! Keevitus 4.5, paagi keevitus kere seest, ?lemine perimeeter, 200+480+200 mm
MoveJ [[1166.72,200.76,754.22],[0.178804,0.624372,-0.674087,0.351848],[1,-1,0,0],[1642.5,-0.000860473,-0.00206977,9E+09,9E+09,9E+09]], v600, z5, tPKI500\WObj:=w7000714;
MoveJ [[768.08,246.74,591.99],[0.154796,0.528852,-0.735934,0.393392],[1,-1,0,0],[1642.5,-10.0074,10.0282,9E+09,9E+09,9E+09]], v600, z5, tPKI500\WObj:=w7000714;
MoveJ [[714.09,147.89,358.50],[0.225232,0.837144,-0.327827,0.375489],[1,0,-1,0],[1642.5,-10.0076,10.0282,9E+09,9E+09,9E+09]], v600, z5, tPKI500\WObj:=w7000714;
ArcLStart [[728.05,133.48,311.58],[0.225215,0.837245,-0.327668,0.375413],[1,0,-1,0],[1642.5,-10.0073,10.0263,9E+09,9E+09,9E+09]], v600, seam1, m178job71, fine, tPKI500\WObj:=w7000714;
ArcL [[731.78,132.97,313.87],[0.240446,0.872935,-0.311321,0.288531],[1,0,-1,0],[1642.5,-10.0064,10.0273,9E+09,9E+09,9E+09]], v600, seam1, m178job71, z5, tPKI500\WObj:=w7000714;
ArcL [[741.60,132.83,314.58],[0.29466,0.908407,-0.270939,0.120687],[1,0,-1,0],[1642.5,-10.0074,10.0279,9E+09,9E+09,9E+09]], v600, seam1, m178job71, z5, tPKI500\WObj:=w7000714;
ArcL [[910.71,134.35,280.92],[0.294691,0.908428,-0.27085,0.120657],[0,0,-2,0],[1642.5,-10.0043,10.0255,9E+09,9E+09,9E+09]], v600, seam1, m178job71, z5, tPKI500\WObj:=w7000714;
ArcL [[922.12,135.61,281.18],[0.279875,0.895951,-0.24893,0.238699],[1,0,-1,0],[1642.5,-10.0074,10.0278,9E+09,9E+09,9E+09]], v600, seam1, m178job71, z5, tPKI500\WObj:=w7000714;
ArcLEnd [[922.62,141.92,281.42],[0.279881,0.895944,-0.248942,0.238705],[1,0,-1,0],[1642.5,-10.0074,10.0275,9E+09,9E+09,9E+09]], v600, seam1, m178job71, fine, tPKI500\WObj:=w7000714;
!
! lisatud wave
! tagant
MoveJ [[875.14,205.61,382.45],[0.279827,0.895934,-0.249016,0.238729],[1,0,-1,0],[1642.5,-10.0075,10.028,9E+09,9E+09,9E+09]], v600, z5, tPKI500\WObj:=w7000714;
! vahetada kiirust v6 v4 peale, sisemis mootori plaadi keevitus.
!Stop;
MoveJ [[865.35,316.77,434.79],[0.116074,-0.918576,0.297867,-0.232427],[1,0,-2,0],[1642.5,-10.0075,10.0279,9E+09,9E+09,9E+09]], v600, z5, tPKI500\WObj:=w7000714;
ArcLStart [[926.89,602.47,281.95],[0.171376,-0.936359,0.129511,-0.277651],[1,0,-2,0],[1642.51,-14.9733,15.0033,9E+09,9E+09,9E+09]], v600, seam1, m178job72, fine, tPKI500\WObj:=w7000714;
ArcL [[926.87,568.08,279.51],[0.00893682,-0.937691,0.124368,-0.324329],[1,0,-2,0],[1642.51,-14.9738,15.0031,9E+09,9E+09,9E+09]], v600, seam1, m178job72, z5, tPKI500\WObj:=w7000714;
ArcL [[925.93,323.18,279.50],[0.0485623,0.933539,-0.130258,0.330425],[1,0,-2,0],[1642.52,-14.972,15.0016,9E+09,9E+09,9E+09]], v600, seam1, m178job72, z5, tPKI500\WObj:=w7000714;
ArcL [[925.26,220.26,279.26],[0.0817255,0.935642,-0.127401,0.31885],[1,0,-2,0],[1642.51,-14.9732,15.0032,9E+09,9E+09,9E+09]], v600, seam1, m178job72, z5, tPKI500\WObj:=w7000714;
ArcLEnd [[923.08,136.67,281.83],[0.114078,0.93955,-0.126756,0.29693],[1,0,-2,0],[1642.51,-14.9734,15.0032,9E+09,9E+09,9E+09]], v600, seam1, m178job72, fine, tPKI500\WObj:=w7000714;
MoveJ [[835.54,241.64,426.42],[0.113929,0.939526,-0.126799,0.297043],[1,0,-2,0],[1642.51,-14.9735,15.0031,9E+09,9E+09,9E+09]], v600, z5, tPKI500\WObj:=w7000714;
!Stop;
!
!
!
!parem serv
MoveJ [[789.61,533.16,507.65],[0.224235,-0.952885,-0.0679482,-0.192649],[1,0,-2,0],[1642.51,-9.95104,-9.97571,9E+09,9E+09,9E+09]], v600, z5, tPKI500\WObj:=w7000714;
MoveJ [[647.14,569.61,433.86],[0.223791,-0.860771,-0.25761,-0.377663],[1,0,-2,0],[1642.51,-9.951,-9.97571,9E+09,9E+09,9E+09]], v600, z5, tPKI500\WObj:=w7000714;
ArcLStart [[727.96,611.07,312.95],[0.295562,-0.83914,-0.288966,-0.353535],[1,0,-2,0],[1642.51,-9.95001,-9.97452,9E+09,9E+09,9E+09]], v600, seam1, m178job71, fine, tPKI500\WObj:=w7000714;
ArcL [[732.79,610.32,317.12],[0.233775,-0.892702,-0.242611,-0.299288],[1,0,-2,0],[1642.51,-9.95127,-9.97524,9E+09,9E+09,9E+09]], v600, seam1, m178job71, z5, tPKI500\WObj:=w7000714;
ArcL [[737.79,609.46,317.60],[0.277417,-0.862841,-0.352886,-0.232418],[1,0,-2,0],[1642.51,-9.951,-9.97587,9E+09,9E+09,9E+09]], v600, seam1, m178job71, z5, tPKI500\WObj:=w7000714;
ArcL [[848.31,608.76,296.63],[0.329544,-0.875695,-0.325912,-0.135432],[1,0,-2,0],[1642.51,-9.95093,-9.97579,9E+09,9E+09,9E+09]], v600, seam1, m178job71, z5, tPKI500\WObj:=w7000714;
ArcL [[912.96,610.64,282.06],[0.338522,-0.884944,-0.249387,-0.200211],[0,0,-2,0],[1642.51,-9.95089,-9.97587,9E+09,9E+09,9E+09]], v600, seam1, m178job71, z5, tPKI500\WObj:=w7000714;
ArcLEnd [[922.77,607.32,283.12],[0.338972,-0.876763,-0.227105,-0.254579],[1,0,-2,0],[1642.51,-9.951,-9.97651,9E+09,9E+09,9E+09]], v600, seam1, m178job71, fine, tPKI500\WObj:=w7000714;
MoveJ [[629.08,382.85,564.19],[0.319673,-0.886676,-0.259097,-0.210916],[1,0,-2,0],[1642.51,-9.95097,-9.97562,9E+09,9E+09,9E+09]], v600, z5, tPKI500\WObj:=w7000714;
!Stop;
MoveJ [[687.39,482.34,438.81],[0.235271,-0.840752,-0.0361746,-0.486288],[1,0,-2,0],[1642.57,-40.0195,-20.0296,9E+09,9E+09,9E+09]], v600, z5, tPKI500\WObj:=w7000714;
MoveJ [[702.69,575.43,343.37],[0.24259,-0.815559,-0.337914,-0.40228],[1,0,-2,0],[1642.57,-40.0195,-20.0295,9E+09,9E+09,9E+09]], v600, z5, tPKI500\WObj:=w7000714;
ArcLStart [[728.60,610.74,312.98],[0.242341,-0.815698,-0.337901,-0.402159],[1,0,-2,0],[1642.57,-40.0167,-20.0299,9E+09,9E+09,9E+09]], v600, seam1, m178job71, fine, tPKI500\WObj:=w7000714;
ArcL [[720.63,611.32,299.17],[0.233436,-0.753089,-0.346163,-0.508466],[1,0,-2,0],[1642.57,-40.0193,-20.0291,9E+09,9E+09,9E+09]], v600, seam1, m178job71, z5, tPKI500\WObj:=w7000714;
ArcL [[687.24,612.19,231.30],[0.233498,-0.753121,-0.346121,-0.508418],[1,0,-2,0],[1642.57,-40.0184,-20.0296,9E+09,9E+09,9E+09]], v600, seam1, m178job71, z5, tPKI500\WObj:=w7000714;
ArcL [[665.17,611.16,193.43],[0.258577,-0.862801,-0.23332,-0.366436],[1,0,-2,0],[1642.57,-40.0177,-20.0296,9E+09,9E+09,9E+09]], v600, seam1, m178job71, z5, tPKI500\WObj:=w7000714;
ArcLEnd [[661.51,603.60,190.16],[0.237634,-0.935104,-0.126943,-0.230211],[1,1,-2,0],[1642.56,-40.0186,-20.0296,9E+09,9E+09,9E+09]], v600, seam1, m178job71, fine, tPKI500\WObj:=w7000714;
!
! lisatud wave
!paagi alumine omblus
!
MoveJ [[549.09,512.65,343.03],[0.23778,-0.935051,-0.126935,-0.230282],[1,1,-2,0],[1642.57,-40.0195,-20.0296,9E+09,9E+09,9E+09]], v600, z5, tPKI500\WObj:=w7000714;
!Stop;
MoveJ [[610.18,311.79,265.60],[0.0869508,-0.984478,-0.0404527,-0.146997],[1,1,-2,0],[1642.58,-30.2802,-29.5527,9E+09,9E+09,9E+09]], v600, z5, tPKI500\WObj:=w7000714;
ArcLStart [[661.41,139.64,189.28],[0.194623,0.960194,-0.0696521,0.18788],[1,1,-2,0],[1642.58,-30.2802,-29.5527,9E+09,9E+09,9E+09]], v600, seam1, m178job72, fine, tPKI500\WObj:=w7000714;
ArcL [[662.37,506.32,187.42],[0.0471849,0.986929,-0.072589,0.135933],[1,1,-2,0],[1642.58,-30.0157,-20.0181,9E+09,9E+09,9E+09]], v600, seam1, m178job72, z5, tPKI500\WObj:=w7000714;
ArcLEnd [[663.45,604.68,191.14],[0.105846,-0.972983,0.037102,-0.201806],[1,1,-2,0],[1642.58,-30.0163,-20.018,9E+09,9E+09,9E+09]], v600, seam1, m178job72, fine, tPKI500\WObj:=w7000714;
!
! lyhike ?mblus
MoveJ [[617.30,284.42,476.03],[0.212151,0.951515,-0.144357,0.16963],[1,1,-2,0],[1642.58,-30.0165,-20.0181,9E+09,9E+09,9E+09]], v600, z5, tPKI500\WObj:=w7000714;
!Stop;
MoveJ [[651.45,220.87,434.81],[0.264842,0.922097,-0.154916,0.235791],[1,0,-2,0],[1933.53,-34.9957,-3.2167,9E+09,9E+09,9E+09]], v600, z5, tPKI500\WObj:=w7000714;
ArcLStart [[728.67,134.77,313.36],[0.30273,0.917485,-0.0333896,0.255856],[1,0,-2,0],[1933.53,-34.9956,-3.21679,9E+09,9E+09,9E+09]], v600, seam1, m178job71, fine, tPKI500\WObj:=w7000714;
ArcL [[724.98,135.31,307.57],[0.302757,0.917479,-0.0333964,0.255845],[1,0,-2,0],[1933.53,-34.9956,-3.21658,9E+09,9E+09,9E+09]], v600, seam1, m178job71, z5, tPKI500\WObj:=w7000714;
ArcL [[671.99,137.01,206.82],[0.302795,0.91747,-0.0334103,0.255828],[1,0,-2,0],[1933.53,-34.9956,-3.21679,9E+09,9E+09,9E+09]], v600, seam1, m178job71, z5, tPKI500\WObj:=w7000714;
ArcL [[664.98,136.99,190.97],[0.302877,0.917453,-0.0334249,0.255792],[1,0,-2,0],[1933.53,-34.9956,-3.21658,9E+09,9E+09,9E+09]], v600, seam1, m178job71, z5, tPKI500\WObj:=w7000714;
ArcLEnd [[664.39,139.97,190.67],[0.302877,0.917455,-0.0334302,0.255786],[1,0,-2,0],[1933.53,-34.9957,-3.21658,9E+09,9E+09,9E+09]], v600, seam1, m178job71, fine, tPKI500\WObj:=w7000714;
MoveJ [[621.65,263.46,419.87],[0.302888,0.917449,-0.0334298,0.255793],[1,0,-2,0],[1933.53,-34.9957,-3.21658,9E+09,9E+09,9E+09]], v600, z5, tPKI500\WObj:=w7000714;

MoveJ [[1209.88,107.35,1002.71],[0.253271,0.875994,-0.262765,0.315348],[0,0,-2,0],[1642.58,-35.0333,19.9774,9E+09,9E+09,9E+09]], v600, z5, tPKI500\WObj:=w7000714;
!Stop;
! viia parandused sisse, kuumem kaar ja nurgad t?ita

! laua p??ramine -50 ja -90 kraadi
MoveJ [[463.28,65.52,1004.63],[0.457365,0.217534,-0.820402,-0.265402],[1,0,-2,0],[1642.51,-50.0165,-90.0065,9E+09,9E+09,9E+09]], v200, z5, tPKI500\WObj:=w7000714;

! Keevitus 4.6, p?hja ?mblus seest, 410+190 mm, paremalt
MoveJ [[196.38,248.72,1103.93],[0.699729,-0.625929,-0.332338,-0.0902487],[1,0,-2,0],[1642.51,-50.0165,-90.0066,9E+09,9E+09,9E+09]], v600, z5, tPKI500\WObj:=w7000714;
MoveJ [[61.15,515.96,761.72],[0.695758,-0.625539,-0.342321,-0.0862556],[1,1,-2,0],[1642.51,-50.0158,-90.0066,9E+09,9E+09,9E+09]], v600, z5, tPKI500\WObj:=w7000714;
MoveJ [[-48.26,518.22,717.52],[0.699706,-0.625962,-0.332322,-0.0902608],[1,1,-2,0],[1642.51,-50.0156,-90.0066,9E+09,9E+09,9E+09]], v600, z5, tPKI500\WObj:=w7000714;
MoveJ [[-178.59,455.25,672.83],[0.499833,-0.795207,-0.343189,0.00592692],[1,1,-2,0],[1642.51,-50.0156,-90.0066,9E+09,9E+09,9E+09]], v600, z5, tPKI500\WObj:=w7000714;
MoveJ [[-180.79,492.80,657.18],[0.521548,-0.780897,-0.342706,-0.0272303],[1,1,-2,0],[1642.51,-53.4217,-90.0073,9E+09,9E+09,9E+09]], v600, z5, tPKI500\WObj:=w7000714;
ArcLStart [[-239.25,512.85,655.67],[0.502988,-0.848154,-0.154897,0.0603867],[1,1,-3,0],[1642.51,-53.4215,-90.0079,9E+09,9E+09,9E+09]], v600, seam1, m178job73, fine, tPKI500\WObj:=w7000714;
!ArcL [[-148.87,554.55,608.87],[0.508794,-0.780118,-0.362131,0.0375068],[1,1,-2,0],[1642.51,-50.0154,-90.0066,9E+09,9E+09,9E+09]], v600, seam1, wld200v6sh14, z5, tPKI500\WObj:=w7000714;
ArcLEnd [[-35.01,617.08,549.75],[0.452558,-0.879456,-0.14001,0.0463462],[1,1,-2,0],[1642.51,-57.3737,-90.0072,9E+09,9E+09,9E+09]], v600, seam1, m178job73, fine, tPKI500\WObj:=w7000714;
MoveL [[53.79,568.86,617.64],[0.452549,-0.879461,-0.140004,0.0463546],[1,1,-2,0],[1642.51,-57.3737,-90.0073,9E+09,9E+09,9E+09]], v600, z5, tPKI500\WObj:=w7000714;
MoveJ [[35.56,572.76,595.15],[0.503916,-0.851326,-0.141306,0.0367077],[1,1,-2,0],[1642.51,-64.1768,-89.8231,9E+09,9E+09,9E+09]], v600, z5, tPKI500\WObj:=w7000714;
ArcLStart [[-26.02,618.24,544.95],[0.43508,-0.890284,-0.119141,0.0625034],[1,1,-2,0],[1642.51,-64.1769,-89.8229,9E+09,9E+09,9E+09]], v600, seam1, m178job73, fine, tPKI500\WObj:=w7000714;
ArcLEnd [[135.95,615.43,462.61],[0.421252,-0.894487,-0.14864,-0.0186384],[1,1,-2,0],[1642.51,-64.1769,-89.8228,9E+09,9E+09,9E+09]], v600, seam1, m178job73, fine, tPKI500\WObj:=w7000714;
MoveJ [[177.09,497.45,621.56],[0.421267,-0.89448,-0.148643,-0.0186307],[1,1,-2,0],[1642.51,-64.1768,-89.823,9E+09,9E+09,9E+09]], v600, z5, tPKI500\WObj:=w7000714;
!Stop;
! liiga palju t?idab, kiirust t?sta

! Keevitus 4.7, p?hja ?mblus seest, 180 mm, paremalt
MoveJ [[404.65,497.01,626.01],[0.429163,-0.845716,-0.305144,-0.0864462],[1,1,-2,0],[1950.19,-50.0155,-90.0066,9E+09,9E+09,9E+09]], v600, z5, tPKI500\WObj:=w7000714;
MoveJ [[512.35,464.70,588.20],[0.429153,-0.845719,-0.305149,-0.0864401],[1,1,-3,0],[1950.19,-50.0155,-90.0065,9E+09,9E+09,9E+09]], v600, z5, tPKI500\WObj:=w7000714;
MoveJ [[519.14,513.74,923.36],[0.398656,-0.898555,-0.0969189,-0.155823],[1,-1,0,0],[1950.19,-50.0155,-90.0065,9E+09,9E+09,9E+09]], v600, z5, tPKI500\WObj:=w7000714;
MoveJ [[461.61,590.34,346.14],[0.436335,-0.892563,-0.0806882,-0.0802135],[1,0,-1,0],[1950.19,-50.0154,-90.0063,9E+09,9E+09,9E+09]], v600, z5, tPKI500\WObj:=w7000714;
ArcLStart [[362.37,616.29,341.75],[0.405567,-0.907589,-0.0994243,-0.0437363],[1,0,-1,0],[1950.19,-50.0155,-90.0064,9E+09,9E+09,9E+09]], v600, seam1, m178job73, fine, tPKI500\WObj:=w7000714;
ArcLEnd [[521.04,611.94,261.93],[0.375808,-0.920622,-0.0997011,-0.0358339],[1,0,-1,0],[1950.19,-50.0155,-90.0071,9E+09,9E+09,9E+09]], v600, seam1, m178job73, fine, tPKI500\WObj:=w7000714;
MoveJ [[520.88,573.24,288.35],[0.346336,-0.937403,-0.0309934,-0.0191679],[1,0,-1,0],[1912.44,-50.0155,-90.0084,9E+09,9E+09,9E+09]], v600, z5, tPKI500\WObj:=w7000714;
ArcLStart [[531.51,613.38,255.56],[0.346292,-0.937416,-0.0310979,-0.0191738],[1,0,-1,0],[1912.44,-50.0155,-90.0083,9E+09,9E+09,9E+09]], v600, seam1, m178job73, fine, tPKI500\WObj:=w7000714;
ArcLEnd [[653.72,608.94,194.33],[0.390845,-0.857992,-0.281743,-0.178077],[1,0,0,0],[1959.61,-55.9377,-89.965,9E+09,9E+09,9E+09]], v600, seam1, m178job73, fine, tPKI500\WObj:=w7000714;
MoveL [[657.28,415.67,487.92],[0.390843,-0.857996,-0.281742,-0.178065],[1,-1,0,0],[1959.61,-55.9377,-89.9649,9E+09,9E+09,9E+09]], v600, z5, tPKI500\WObj:=w7000714;

GOTO paagiall;

! Keevitus 4.8, paagi ?mblus seest, ?lalt-alla, 150 mm, paremalt
MoveJ [[708.82,589.48,349.92],[0.26351,-0.882482,-0.294377,-0.25521],[1,1,-2,0],[1950.19,-50.0147,-90.0062,9E+09,9E+09,9E+09]], v600, z5, tPKI500\WObj:=w7000714;
ArcLStart [[732.29,612.15,312.42],[0.263422,-0.882509,-0.294419,-0.255159],[1,1,-2,0],[1950.19,-50.0147,-90.0062,9E+09,9E+09,9E+09]], v600, seam1, wld100v4sh16, fine, tPKI500\WObj:=w7000714;
ArcL [[721.14,612.59,306.41],[0.263365,-0.882522,-0.294466,-0.255117],[1,1,-2,0],[1950.19,-50.0148,-90.0059,9E+09,9E+09,9E+09]], v600, seam1, wld100v4sh16, z5, tPKI500\WObj:=w7000714;
ArcLEnd [[660.86,607.69,192.53],[0.282267,-0.873646,-0.270174,-0.289957],[1,1,-2,0],[1950.19,-50.0148,-90.0062,9E+09,9E+09,9E+09]], v600, seam1, wld100v4sh16, fine, tPKI500\WObj:=w7000714;
MoveJ [[659.87,534.23,289.89],[0.282313,-0.873638,-0.270157,-0.289951],[1,1,-2,0],[1950.19,-50.0147,-90.0062,9E+09,9E+09,9E+09]], v600, z5, tPKI500\WObj:=w7000714;
MoveJ [[656.91,166.38,784.04],[0.282307,-0.87364,-0.27016,-0.289949],[1,0,-1,0],[1950.19,-50.0147,-90.0062,9E+09,9E+09,9E+09]], v600, z5, tPKI500\WObj:=w7000714;
MoveJ [[655.16,-102.11,1008.14],[0.282304,-0.87364,-0.27016,-0.289954],[1,0,-1,0],[1950.19,-50.0147,-90.0061,9E+09,9E+09,9E+09]], v600, z5, tPKI500\WObj:=w7000714;
! liiga palju t?idab, kiirust t?sta

paagiall:

! laua p??ramine 50 ja -90 kraadi
MoveJ [[629.05,106.87,1333.63],[0.742615,-0.0488617,-0.662818,0.0825176],[1,0,-2,0],[1950.19,-50.0144,-90.0065,9E+09,9E+09,9E+09]], v600, z5, tPKI500\WObj:=w7000714;
MoveJ [[666.24,1407.62,346.58],[0.485843,0.779341,0.394853,-0.0260103],[1,0,-1,0],[1950.2,49.9779,-90.0059,9E+09,9E+09,9E+09]], v200, z5, tPKI500\WObj:=w7000714;

! Keevitus 4.9, p?hja ?mblus seest, 410+190 mm, vasakult
MoveJ [[388.60,678.79,1213.60],[0.557133,0.824872,0.0604223,0.0744247],[0,0,-1,0],[12.7994,49.9779,-90.0058,9E+09,9E+09,9E+09]], v600, z5, tPKI500\WObj:=w7000714;
MoveJ [[384.49,294.23,786.50],[0.557145,0.824863,0.0604211,0.074436],[0,0,-1,0],[12.7984,49.978,-90.0056,9E+09,9E+09,9E+09]], v600, z5, tPKI500\WObj:=w7000714;
MoveJ [[65.60,161.93,784.24],[0.484927,0.853835,-0.0416443,-0.184603],[0,1,-2,0],[12.7988,49.978,-90.0056,9E+09,9E+09,9E+09]], v600, z5, tPKI500\WObj:=w7000714;
MoveJ [[-229.88,281.25,701.83],[0.48494,0.85383,-0.0416313,-0.184598],[0,1,-2,0],[12.7988,49.978,-90.0056,9E+09,9E+09,9E+09]], v600, z5, tPKI500\WObj:=w7000714;
ArcLStart [[-229.82,242.03,655.30],[0.485298,0.853687,-0.0412593,-0.184401],[0,1,-2,0],[12.7994,49.9782,-90.0049,9E+09,9E+09,9E+09]], v600, seam1, m178job75, fine, tPKI500\WObj:=w7000714;
ArcL [[-84.08,165.89,578.50],[0.498551,0.849644,-0.0346232,-0.16839],[0,1,-2,0],[12.7972,49.9796,-90.004,9E+09,9E+09,9E+09]], v600, seam1, m178job75, z5, tPKI500\WObj:=w7000714;
ArcL [[-27.66,140.23,549.05],[0.527487,0.84556,-0.00876734,-0.0819137],[0,1,-2,0],[12.7972,49.9795,-90.0041,9E+09,9E+09,9E+09]], v600, seam1, m178job75, z5, tPKI500\WObj:=w7000714;
ArcL [[16.72,138.82,525.36],[0.481758,0.871608,-0.0848704,-0.0317208],[0,1,-2,0],[12.7933,49.9797,-90.0036,9E+09,9E+09,9E+09]], v600, seam1, m178job75, z5, tPKI500\WObj:=w7000714;
ArcLEnd [[133.70,138.04,464.64],[0.451188,0.883091,-0.127052,0.0209757],[0,2,-2,0],[12.7949,49.9799,-90.0038,9E+09,9E+09,9E+09]], v600, seam1, m178job73, fine, tPKI500\WObj:=w7000714;
MoveJ [[136.36,209.25,580.64],[0.468487,0.870946,-0.136243,-0.0584185],[0,1,-2,0],[12.7984,49.978,-90.0055,9E+09,9E+09,9E+09]], v600, z5, tPKI500\WObj:=w7000714;
! liiga palju t?idab, kiirust t?sta

! Keevitus 4.10, sarniiri k?rv pealt, 100+50, vasakult
MoveJ [[-36.62,215.87,637.30],[0.532452,0.822587,-0.164204,-0.113512],[0,1,-2,0],[12.8001,49.9781,-90.0053,9E+09,9E+09,9E+09]], v600, z5, tPKI500\WObj:=w7000714;
ArcLStart [[-77.82,169.87,614.91],[0.492202,0.845085,-0.126744,-0.165852],[0,1,-2,0],[12.8004,49.9783,-90.0044,9E+09,9E+09,9E+09]], v600, seam1, m178job75, fine, tPKI500\WObj:=w7000714;
ArcL [[-14.48,137.24,582.80],[0.468789,0.86953,-0.05854,-0.143978],[0,1,-2,0],[12.8017,49.9785,-90.005,9E+09,9E+09,9E+09]], v600, seam1, m178job75, z5, tPKI500\WObj:=w7000714;
ArcLEnd [[24.32,136.30,561.78],[0.4688,0.869526,-0.0585137,-0.143972],[0,1,-2,0],[12.8017,49.9783,-90.0048,9E+09,9E+09,9E+09]], v600, seam1, m178job75, fine, tPKI500\WObj:=w7000714;
MoveJ [[26.28,211.80,629.17],[0.53258,0.822524,-0.164103,-0.11351],[0,1,-2,0],[12.8001,49.9781,-90.0056,9E+09,9E+09,9E+09]], v600, z5, tPKI500\WObj:=w7000714;
MoveJ [[454.07,297.49,698.34],[0.532584,0.822521,-0.164102,-0.113513],[0,1,-2,0],[12.8001,49.978,-90.0054,9E+09,9E+09,9E+09]], v600, z5, tPKI500\WObj:=w7000714;
! liiga kuum

! Keevitus 4.11, p?hja ?mblus seest, 180 mm, vasakult
MoveJ [[462.46,181.06,454.07],[0.532569,0.822509,-0.164117,-0.113651],[0,1,-2,0],[12.7994,49.9781,-90.0054,9E+09,9E+09,9E+09]], v600, z5, tPKI500\WObj:=w7000714;
MoveJ [[373.51,148.16,352.75],[0.532701,0.836564,-0.127494,0.0116893],[0,1,-2,0],[12.8004,49.9782,-90.0053,9E+09,9E+09,9E+09]], v600, z5, tPKI500\WObj:=w7000714;
ArcLStart [[363.62,133.40,339.74],[0.385285,0.913722,-0.128687,-0.0104206],[0,1,-3,0],[12.8033,49.9784,-90.0053,9E+09,9E+09,9E+09]], v600, seam1, m178job73, fine, tPKI500\WObj:=w7000714;
ArcLEnd [[521.63,134.33,258.78],[0.384893,0.913779,-0.129338,-0.0118155],[0,1,-2,0],[12.804,49.978,-90.0048,9E+09,9E+09,9E+09]], v600, seam1, m178job73, fine, tPKI500\WObj:=w7000714;
MoveJ [[529.89,336.50,401.69],[0.385019,0.91381,-0.12889,-0.00995835],[0,1,-2,0],[12.8004,49.9781,-90.0051,9E+09,9E+09,9E+09]], v600, z5, tPKI500\WObj:=w7000714;
MoveJ [[533.43,251.88,352.38],[0.378148,0.919534,-0.10133,0.0345688],[0,1,-2,0],[12.8017,49.9784,-90.005,9E+09,9E+09,9E+09]], v600, z5, tPKI500\WObj:=w7000714;
ArcLStart [[531.13,134.57,252.75],[0.378146,0.919534,-0.101345,0.0345315],[0,1,-2,0],[12.8017,49.9784,-90.005,9E+09,9E+09,9E+09]], v600, seam1, m178job73, fine, tPKI500\WObj:=w7000714;
ArcLEnd [[657.61,136.14,189.32],[0.303811,0.940087,-0.0293689,0.151901],[0,1,-3,0],[12.7988,49.9785,-90.0046,9E+09,9E+09,9E+09]], v600, seam1, m178job73, fine, tPKI500\WObj:=w7000714;
MoveL [[549.64,239.77,442.99],[0.323521,0.93805,-0.0571311,0.110153],[0,1,-3,0],[12.7994,49.9786,-90.005,9E+09,9E+09,9E+09]], v600, z5, tPKI500\WObj:=w7000714;

MoveJ [[730.99,435.16,896.64],[0.414132,0.875986,-0.0952889,0.228177],[0,-1,0,0],[12.8004,49.9782,-90.0052,9E+09,9E+09,9E+09]], v600, z5, tPKI500\WObj:=w7000714;
MoveJ [[630.56,205.75,1267.74],[0.0352222,0.637589,0.698102,-0.323875],[1,0,-2,0],[63.5912,90.0341,-90.0151,9E+09,9E+09,9E+09]], v600, z5, tPKI500\WObj:=w7000714;

! laua p??ramine 90 ja -90 kraadi
MoveJ [[628.71,206.23,996.67],[0.0352126,0.637586,0.698102,-0.32388],[1,0,-2,0],[334.665,90.0341,-90.0152,9E+09,9E+09,9E+09]], v200, z5, tPKI500\WObj:=w7000714;
MoveJ [[897.19,986.56,937.18],[0.846952,0.13011,-0.222738,0.464901],[1,-1,1,0],[1328.03,90.034,-90.0145,9E+09,9E+09,9E+09]], v200, z5, tPKI500\WObj:=w7000714;
MoveJ [[1264.54,861.62,340.94],[0.846954,0.130102,-0.222719,0.464908],[1,-1,2,0],[1328.03,90.0341,-90.0147,9E+09,9E+09,9E+09]], v200, z5, tPKI500\WObj:=w7000714;

! Keevitus 4.19, tagumine kereplaat, l?hike ?mblus, 30 mm, paremalt, OK
MoveJ [[1033.09,580.58,354.82],[0.686293,0.0368718,-0.42949,-0.585817],[1,-1,-1,0],[2188.28,-90.0189,-90.0141,9E+09,9E+09,9E+09]], v600, z5, tPKI500\WObj:=w7000714;
MoveJ [[979.14,569.48,388.43],[0.806601,-0.0278027,-0.197946,-0.556273],[1,-1,0,0],[2188.28,-90.0189,-90.0141,9E+09,9E+09,9E+09]], v600, z5, tPKI500\WObj:=w7000714;
ArcLStart [[978.92,568.70,409.45],[0.806531,-0.0276883,-0.198257,-0.55627],[1,-1,0,0],[2188.28,-90.0187,-90.0134,9E+09,9E+09,9E+09]], v600, seam1, m178job74, fine, tPKI500\WObj:=w7000714;
ArcLEnd [[979.79,595.48,407.03],[0.806541,-0.0276795,-0.198221,-0.556269],[1,-1,0,0],[2188.28,-90.0191,-90.0136,9E+09,9E+09,9E+09]], v600, seam1, m178job74, fine, tPKI500\WObj:=w7000714;
MoveL [[991.84,562.72,392.18],[0.806551,-0.0277066,-0.198182,-0.556268],[1,-1,0,0],[2188.28,-90.0181,-90.0139,9E+09,9E+09,9E+09]], v600, z5, tPKI500\WObj:=w7000714;
MoveJ [[984.53,239.20,388.90],[0.844678,0.202999,-0.0676416,-0.49065],[1,-1,-1,0],[2188.28,-90.0188,-90.0142,9E+09,9E+09,9E+09]], v600, z5, tPKI500\WObj:=w7000714;
ArcLStart [[975.41,149.41,410.22],[0.844693,0.203001,-0.0678212,-0.490598],[1,-1,-1,0],[2188.28,-90.018,-90.0166,9E+09,9E+09,9E+09]], v600, seam1, m178job74, fine, tPKI500\WObj:=w7000714;
ArcLEnd [[974.88,173.69,411.07],[0.844673,0.203034,-0.0678784,-0.49061],[1,-1,-1,0],[2188.28,-90.0188,-90.0144,9E+09,9E+09,9E+09]], v600, seam1, m178job74, fine, tPKI500\WObj:=w7000714;
MoveJ [[1127.32,173.99,318.93],[0.844677,0.203007,-0.0677125,-0.490637],[1,-1,-1,0],[2188.28,-90.0188,-90.0143,9E+09,9E+09,9E+09]], v600, z5, tPKI500\WObj:=w7000714;
MoveJ [[1123.72,259.36,389.60],[0.806585,-0.0277724,-0.198013,-0.556274],[1,-1,-1,0],[2188.28,-90.0189,-90.014,9E+09,9E+09,9E+09]], v600, z5, tPKI500\WObj:=w7000714;
MoveJ [[1120.90,-120.19,388.59],[0.806586,-0.0277689,-0.198012,-0.556274],[1,-1,-1,0],[2188.28,-90.019,-90.014,9E+09,9E+09,9E+09]], v600, z5, tPKI500\WObj:=w7000714;
MoveJ [[1027.41,-315.13,387.66],[0.806588,-0.0277633,-0.198009,-0.556273],[1,-1,-1,0],[2188.28,-90.019,-90.0141,9E+09,9E+09,9E+09]], v600, z5, tPKI500\WObj:=w7000714;
MoveJ [[1587.39,-314.57,2238.78],[0.395106,-0.543248,0.72299,-0.16143],[0,-1,-1,0],[2188.28,-90.0189,-90.0141,9E+09,9E+09,9E+09]], v600, z5, tPKI500\WObj:=w7000714;

! laua p??ramine 0 ja 0 kraadi
MoveJ [[2571.99,-849.77,725.34],[0.516673,0.188187,-0.752202,0.36308],[0,-1,-1,0],[2188.28,-0.0178089,-0.0101717,9E+09,9E+09,9E+09]], v200, z5, tPKI500\WObj:=w7000714;
MoveJ [[1078.51,394.47,809.90],[0.143804,-0.871177,0.456961,-0.107516],[1,-1,0,0],[2188.28,-0.0178089,-0.0101295,9E+09,9E+09,9E+09]], v600, z5, tPKI500\WObj:=w7000714;
MoveL [[784.81,404.00,996.38],[0.219819,-0.844688,0.418448,-0.251165],[1,-1,0,0],[2188.28,-19.3919,-1.07477,9E+09,9E+09,9E+09]], v600, z5, tPKI500\WObj:=w7000714;
MoveL [[830.09,498.09,533.40],[0.157013,-0.745399,0.376549,-0.5272],[1,-1,0,0],[2188.28,-33.0668,-1.07519,9E+09,9E+09,9E+09]], v600, z5, tPKI500\WObj:=w7000714;
ArcLStart [[968.89,134.51,399.97],[0.229202,0.70512,-0.224113,0.632493],[1,0,-1,0],[2188.27,-33.0655,-1.07654,9E+09,9E+09,9E+09]], v200, seam1, m178job77, fine, tPKI500\WObj:=w7000714;
ArcL [[932.09,135.02,326.61],[0.229208,0.705135,-0.224106,0.632476],[1,0,-1,0],[2188.27,-33.0655,-1.07633,9E+09,9E+09,9E+09]], v200, seam1, m178job77, fine, tPKI500\WObj:=w7000714;
ArcL [[924.27,137.56,288.65],[0.285048,0.869977,-0.140228,0.377128],[1,0,-2,0],[2188.27,-33.0647,-1.07713,9E+09,9E+09,9E+09]], v200, seam1, m178job77, fine, tPKI500\WObj:=w7000714;
ArcLEnd [[916.79,146.87,290.75],[0.225012,0.93026,-0.175906,0.230313],[1,1,-2,0],[2188.27,-33.0647,-1.07692,9E+09,9E+09,9E+09]], v200, seam1, m178job77, fine, tPKI500\WObj:=w7000714;
MoveL [[860.28,390.12,368.97],[0.0097858,0.933264,-0.105499,0.343212],[1,0,-2,0],[2188.27,-33.0647,-1.07705,9E+09,9E+09,9E+09]], v200, fine, tPKI500\WObj:=w7000714;
ArcLStart [[966.40,607.71,401.95],[0.309024,-0.838606,-0.190201,-0.406287],[1,0,-2,0],[2188.27,-33.0639,-1.07755,9E+09,9E+09,9E+09]], v200, seam1, m178job77, fine, tPKI500\WObj:=w7000714;
ArcL [[930.19,608.39,328.98],[0.308956,-0.838652,-0.190164,-0.406262],[1,0,-2,0],[2188.27,-33.0639,-1.07776,9E+09,9E+09,9E+09]], v200, seam1, m178job77, fine, tPKI500\WObj:=w7000714;
ArcL [[923.99,606.70,286.47],[0.284962,-0.883566,-0.155473,-0.337548],[1,1,-2,0],[2188.27,-33.0634,-1.07882,9E+09,9E+09,9E+09]], v200, seam1, m178job77, fine, tPKI500\WObj:=w7000714;
ArcLEnd [[922.74,604.55,283.86],[0.225597,-0.927343,-0.17685,-0.240556],[1,1,-2,0],[2188.27,-33.0634,-1.07882,9E+09,9E+09,9E+09]], v200, seam1, m178job77, fine, tPKI500\WObj:=w7000714;
MoveL [[766.07,413.97,534.40],[0.285128,-0.883476,-0.155522,-0.337618],[1,0,-2,0],[2188.27,-33.0637,-1.07827,9E+09,9E+09,9E+09]], v600, fine, tPKI500\WObj:=w7000714;
MoveL [[1931.24,112.08,1797.85],[0.481099,-0.603835,0.414467,-0.481815],[0,0,-2,0],[2188.27,-33.0635,-1.07827,9E+09,9E+09,9E+09]], v600, fine, tPKI500\WObj:=w7000714;
! laua p??ramine 0 ja 180 kraadi
!MoveJ [[-1805.19,1600.36,726.17],[0.363056,-0.752319,-0.188029,-0.516579],[0,-1,-1,0],[2188.34,-0.0394387,180.004,9E+09,9E+09,9E+09]], v500, z5, tPKI500\WObj:=w7000714;
! laua p??ramine -40 ja 180 kraadi
!MoveJ [[-842.65,1593.50,1984.19],[0.407518,-0.88328,-0.0499407,-0.226392],[0,-1,-1,0],[2188.34,-40.3394,179.976,9E+09,9E+09,9E+09]], v200, z5, tPKI500\WObj:=w7000714;
!MoveJ [[-361.88,238.65,1366.99],[0.233905,-0.220588,-0.921934,0.216031],[0,0,-2,0],[2188.34,-34.9738,179.976,9E+09,9E+09,9E+09]], v600, z5, tPKI500\WObj:=w7000714;
!MoveJ [[-329.76,347.68,853.85],[0.171568,-0.037775,-0.971091,0.161622],[0,1,-2,0],[2188.34,-33.8713,179.976,9E+09,9E+09,9E+09]], v600, z5, tPKI500\WObj:=w7000714;
!ArcLStart [[-267.00,283.63,772.23],[0.159657,0.0398007,-0.944889,0.283041],[1,1,-2,0],[2188.34,-33.8711,179.976,9E+09,9E+09,9E+09]], v600, seam1, wld100v4sh16, fine, tPKI500\WObj:=w7000714;
!ArcLEnd [[-319.65,311.33,800.44],[0.159636,0.0398197,-0.944893,0.283035],[1,1,-2,0],[2188.34,-33.8713,179.976,9E+09,9E+09,9E+09]], v600, seam1, wld100v4sh16, fine, tPKI500\WObj:=w7000714;
!ArcLStart [[-267.16,284.07,771.57],[0.159658,0.0398083,-0.944881,0.283064],[1,1,-2,0],[2188.34,-33.871,179.976,9E+09,9E+09,9E+09]], v600, seam1, wld100v4sh16\Weave:=weave4, fine, tPKI500\WObj:=w7000714;
!ArcLEnd [[-321.12,312.86,800.70],[0.159639,0.0398143,-0.944893,0.283037],[1,1,-2,0],[2188.34,-33.8713,179.976,9E+09,9E+09,9E+09]], v600, seam1, wld100v4sh16\Weave:=weave4, fine, tPKI500\WObj:=w7000714;
!MoveL [[-422.53,369.77,925.81],[0.146248,0.0635872,-0.986461,-0.0382709],[0,0,-2,0],[2188.34,-33.8712,179.976,9E+09,9E+09,9E+09]], v600, fine, tPKI500\WObj:=w7000714;
!MoveL [[-371.17,402.53,866.35],[0.159991,-0.0776618,-0.933329,-0.311882],[0,0,-2,0],[2188.34,-33.8712,179.976,9E+09,9E+09,9E+09]], v600, fine, tPKI500\WObj:=w7000714;
!ArcLStart [[-264.44,468.19,771.49],[0.202364,-0.212347,-0.926323,-0.236398],[1,0,-2,0],[2188.34,-33.8711,179.976,9E+09,9E+09,9E+09]], v600, seam1, wld100v4sh16, fine, tPKI500\WObj:=w7000714;
!ArcLEnd [[-317.75,442.56,798.65],[0.20235,-0.212334,-0.926323,-0.236423],[1,0,-2,0],[2188.34,-33.8711,179.976,9E+09,9E+09,9E+09]], v600, seam1, wld100v4sh16, fine, tPKI500\WObj:=w7000714;
!ArcLStart [[-265.35,467.62,772.88],[0.20236,-0.212345,-0.926325,-0.236395],[1,0,-2,0],[2188.34,-33.8711,179.976,9E+09,9E+09,9E+09]], v600, seam1, wld100v4sh16\Weave:=weave4, fine, tPKI500\WObj:=w7000714;
!ArcLEnd [[-318.74,440.66,800.16],[0.202349,-0.212327,-0.926327,-0.236414],[1,0,-2,0],[2188.34,-33.871,179.976,9E+09,9E+09,9E+09]], v600, seam1, wld100v4sh16\Weave:=weave4, fine, tPKI500\WObj:=w7000714;
!MoveL [[-386.39,410.04,858.22],[0.20235,-0.21233,-0.926323,-0.236427],[0,0,-2,0],[2188.34,-33.8711,179.976,9E+09,9E+09,9E+09]], v600, fine, tPKI500\WObj:=w7000714;
!MoveJ [[-350.68,416.29,1470.07],[0.202358,-0.212326,-0.92632,-0.236433],[0,0,-1,0],[2188.34,-33.8711,179.976,9E+09,9E+09,9E+09]], v600, fine, tPKI500\WObj:=w7000714;
MoveJ [[2571.99,-849.77,725.34],[0.516675,0.188183,-0.752204,0.363076],[0,-1,-1,0],[2188.28,-0.0178089,-0.0101717,9E+09,9E+09,9E+09]], v400, fine, tPKI500\WObj:=w7000714;



! aeg manualis 15:30, 100 % juures


MoveJ mooduli_vahetus, v600, z50, tPKI500\WObj:=w7000714;

ENDPROC


! V?ljast kinnitused ja alt puksid
PROC Seest_alt()

MoveJ mooduli_vahetus, v600, z50, tPKI500\WObj:=w7000714;

!laua liikumine
!Stop;
! Keevitus 5.1, esimene vasak klots ulevalt ja korvalt.
MoveJ [[-290.14,770.26,1028.88],[0.179367,-0.475167,0.667996,-0.5439],[0,0,-1,0],[1372.29,-65.3529,37.4059,9E+09,9E+09,9E+09]], v200, z50, tPKI500\WObj:=w7000714;
MoveJ [[-43.63,789.96,1015.82],[0.0154596,0.0805408,0.981036,-0.175623],[0,-1,0,0],[1372.29,-65.3519,37.4059,9E+09,9E+09,9E+09]], v600, z50, tPKI500\WObj:=w7000714;
ArcLStart [[-30.35,722.48,992.87],[0.0308617,0.0919503,-0.954938,0.280513],[0,0,0,0],[1372.28,-65.3461,37.4041,9E+09,9E+09,9E+09]], v600, seam1, m178job76, fine, tPKI500\WObj:=w7000714;
ArcL [[4.24,779.21,976.32],[0.031198,0.0916798,-0.954822,0.280957],[0,0,0,0],[1372.3,-65.3486,37.4052,9E+09,9E+09,9E+09]], v600, seam1, m178job76, z50, tPKI500\WObj:=w7000714;
ArcL [[4.75,783.75,972.21],[0.163165,0.328816,-0.70964,0.60139],[0,0,-1,0],[1372.29,-65.3489,37.4059,9E+09,9E+09,9E+09]], v600, seam1, m178job76, z50, tPKI500\WObj:=w7000714;
ArcL [[-106.57,785.87,753.86],[0.206514,0.412137,-0.564809,0.684461],[1,0,-1,0],[1372.28,-65.3395,37.4003,9E+09,9E+09,9E+09]], v600, seam1, m178job76, z50, tPKI500\WObj:=w7000714;
ArcL [[-111.66,783.39,751.13],[0.0614244,0.527208,-0.229631,0.815812],[1,0,-1,0],[1372.28,-65.3501,37.4051,9E+09,9E+09,9E+09]], v600, seam1, m178job76, z50, tPKI500\WObj:=w7000714;
ArcLEnd [[-145.83,729.02,766.75],[0.118602,0.614006,-0.031797,0.779692],[1,0,-2,0],[1372.29,-65.3478,37.4021,9E+09,9E+09,9E+09]], v600, seam1, m178job76, fine, tPKI500\WObj:=w7000714;
MoveJ [[-215.14,772.76,801.30],[0.102061,0.714158,0.0425608,0.691196],[1,0,-2,0],[1372.29,-65.3521,37.4058,9E+09,9E+09,9E+09]], v600, z50, tPKI500\WObj:=w7000714;
MoveJ [[-208.50,762.42,1040.05],[0.137789,-0.773479,0.148928,-0.600471],[0,0,-2,0],[1372.29,-65.3521,37.4056,9E+09,9E+09,9E+09]], v600, z50, tPKI500\WObj:=w7000714;
ArcLStart [[-30.79,723.95,992.18],[0.136855,-0.804117,0.0864458,-0.57201],[0,0,-2,0],[1372.29,-65.3435,37.4035,9E+09,9E+09,9E+09]], v600, seam1, m178job76, fine, tPKI500\WObj:=w7000714;
ArcLEnd [[-145.93,726.55,773.14],[0.136768,-0.804096,0.0862477,-0.57209],[0,0,-2,0],[1372.29,-65.3446,37.4062,9E+09,9E+09,9E+09]], v600, seam1, m178job76, fine, tPKI500\WObj:=w7000714;
MoveJ [[-373.93,893.47,896.85],[0.138032,-0.80362,0.0855156,-0.572565],[0,0,-2,0],[1372.29,-65.3521,37.4057,9E+09,9E+09,9E+09]], v600, z50, tPKI500\WObj:=w7000714;




! Keevitus 5.3, p?rkeraua klots parem, esimene ?mblus, pealt ja kuljelt
MoveJ [[-174.00,-345.05,357.08],[0.250849,-0.133618,-0.812081,-0.509653],[1,0,-2,0],[1372.29,-65.4717,-36.1497,9E+09,9E+09,9E+09]], v200, z50, tPKI500\WObj:=w7000714;
MoveJ [[-10.19,-84.76,986.05],[0.275118,-0.267366,-0.642243,-0.66359],[0,0,-2,0],[1372.29,-65.4717,-36.1497,9E+09,9E+09,9E+09]], v600, z50, tPKI500\WObj:=w7000714;
ArcLStart [[-5.29,-25.23,972.07],[0.269578,-0.358495,-0.567203,-0.690718],[0,0,-2,0],[1372.33,-65.4684,-36.1495,9E+09,9E+09,9E+09]], v600, seam1, m178job76, fine, tPKI500\WObj:=w7000714;
ArcL [[-118.04,-25.80,755.94],[0.253515,-0.440375,-0.485319,-0.711524],[1,0,-2,0],[1372.28,-65.4664,-36.1515,9E+09,9E+09,9E+09]], v600, seam1, m178job76, z50, tPKI500\WObj:=w7000714;
ArcL [[-122.46,-23.08,751.12],[0.364637,-0.582226,0.0124595,-0.726566],[1,0,-1,0],[1372.3,-65.4709,-36.1507,9E+09,9E+09,9E+09]], v600, seam1, m178job76, z50, tPKI500\WObj:=w7000714;
ArcL [[-153.48,32.59,768.13],[0.37674,-0.591162,0.132537,-0.700736],[1,0,-1,0],[1372.29,-65.4696,-36.1466,9E+09,9E+09,9E+09]], v600, seam1, m178job76, z50, tPKI500\WObj:=w7000714;
ArcL [[-152.80,36.92,774.93],[0.372014,-0.520105,0.662343,-0.390384],[1,-1,0,0],[1372.29,-65.4622,-36.1483,9E+09,9E+09,9E+09]], v600, seam1, m178job76, z50, tPKI500\WObj:=w7000714;
ArcL [[-39.28,36.72,991.14],[0.345262,-0.453792,0.773924,-0.275519],[1,-1,0,0],[1372.3,-65.4589,-36.1523,9E+09,9E+09,9E+09]], v600, seam1, m178job76, z50, tPKI500\WObj:=w7000714;
ArcL [[-35.16,32.79,991.93],[0.248259,-0.27299,0.925404,0.0864419],[1,-1,0,0],[1372.28,-65.4618,-36.1461,9E+09,9E+09,9E+09]], v600, seam1, m178job76, z50, tPKI500\WObj:=w7000714;
ArcLEnd [[-4.28,-21.64,975.36],[0.137343,-0.249955,0.927968,0.239868],[1,-1,1,0],[1372.29,-65.4709,-36.1483,9E+09,9E+09,9E+09]], v600, seam1, m178job76, fine, tPKI500\WObj:=w7000714;
MoveJ [[-61.03,-65.95,1001.68],[0.133904,-0.241825,0.927325,0.252308],[1,-1,1,0],[1372.29,-65.4722,-36.1495,9E+09,9E+09,9E+09]], v600, z50, tPKI500\WObj:=w7000714;


! Keevitus 5.4, p?rkeraua klots paremalt, teine ?mblus, kuljelt.


! Keevitus 5.5, p?rkeraua klots tagant1, O ?mblus, vasakult
MoveJ [[1208.50,-67.48,645.00],[0.55081,-0.741965,0.19537,0.328526],[0,-1,0,0],[1289.08,-105.992,-131.558,9E+09,9E+09,9E+09]], v200, z50, tPKI500\WObj:=w7000714;
MoveJ [[878.05,-71.80,532.67],[0.377928,-0.771852,0.343338,0.378859],[0,-1,0,0],[1289.08,-105.992,-131.558,9E+09,9E+09,9E+09]], v600, z50, tPKI500\WObj:=w7000714;
ArcLStart [[911.48,1.66,499.56],[0.180122,-0.806357,0.321968,0.462258],[0,-1,1,0],[1289.09,-105.99,-131.558,9E+09,9E+09,9E+09]], v600, seam1, m178job76, fine, tPKI500\WObj:=w7000714;
ArcL [[866.81,-37.76,522.04],[0.241931,-0.80225,0.32882,0.435596],[0,-1,0,0],[1289.08,-105.992,-131.558,9E+09,9E+09,9E+09]], v600, seam1, m178job76, z50, tPKI500\WObj:=w7000714;
ArcL [[859.31,-43.24,520.79],[0.656383,-0.696913,0.229608,0.175374],[0,-1,0,0],[1289.08,-105.991,-131.558,9E+09,9E+09,9E+09]], v600, seam1, m178job76, z50, tPKI500\WObj:=w7000714;
ArcL [[749.03,-43.15,305.63],[0.666588,-0.691289,0.223493,0.16683],[1,-1,0,0],[1289.08,-105.991,-131.558,9E+09,9E+09,9E+09]], v600, seam1, m178job76, z50, tPKI500\WObj:=w7000714;
ArcL [[748.23,-38.21,296.26],[0.881837,-0.46223,0.0260185,-0.0896109],[1,0,-1,0],[1289.08,-105.992,-131.558,9E+09,9E+09,9E+09]], v600, seam1, m178job76, z50, tPKI500\WObj:=w7000714;
ArcLEnd [[795.12,2.54,270.09],[0.92494,-0.290166,-0.143809,-0.199024],[1,0,-1,0],[1289.08,-105.991,-131.558,9E+09,9E+09,9E+09]], v600, seam1, m178job76, fine, tPKI500\WObj:=w7000714;
MoveL [[821.17,-27.30,258.63],[0.924935,-0.290173,-0.143812,-0.199036],[1,0,-1,0],[1289.08,-105.991,-131.558,9E+09,9E+09,9E+09]], v400, z50, tPKI500\WObj:=w7000714;
MoveL [[823.25,-19.25,258.87],[0.774205,0.152692,-0.382226,-0.480829],[1,0,-2,0],[1289.08,-105.991,-131.56,9E+09,9E+09,9E+09]], v400, z50, tPKI500\WObj:=w7000714;
ArcLStart [[801.74,5.40,268.33],[0.774207,0.152706,-0.382226,-0.480821],[1,0,-2,0],[1289.08,-105.991,-131.56,9E+09,9E+09,9E+09]], v600, seam1, m178job76, fine, tPKI500\WObj:=w7000714;
ArcL [[805.46,3.98,276.41],[0.77421,0.152731,-0.382224,-0.480811],[1,0,-2,0],[1289.08,-105.992,-131.559,9E+09,9E+09,9E+09]], v600, seam1, m178job76, z50, tPKI500\WObj:=w7000714;
ArcLEnd [[913.95,3.05,493.11],[0.74603,0.191483,-0.397811,-0.498518],[0,0,-2,0],[1289.08,-105.991,-131.558,9E+09,9E+09,9E+09]], v600, seam1, m178job76, fine, tPKI500\WObj:=w7000714;
MoveJ [[1036.00,-137.14,436.44],[0.829926,0.0635067,-0.342982,-0.435379],[0,0,-2,0],[1289.08,-105.992,-131.558,9E+09,9E+09,9E+09]], v600, z50, tPKI500\WObj:=w7000714;
MoveJ [[771.13,-196.57,635.64],[0.451534,0.540448,-0.297667,-0.644538],[0,-1,-3,0],[1289.08,-106.644,-125.692,9E+09,9E+09,9E+09]], v600, z50, tPKI500\WObj:=w7000714;


! Keevitus 5.6, p?rkeraua klots tagant2, O ?mblus, vasakult
MoveJ [[617.87,726.47,902.15],[0.207025,-0.863971,-0.0872424,-0.45065],[1,-1,-1,0],[931.999,2.9016,-87.1854,9E+09,9E+09,9E+09]], v200, z50, tPKI500\WObj:=w7000714;
MoveJ [[938.69,1079.18,390.78],[0.956989,0.0513518,-0.248038,0.14147],[1,-1,1,0],[652.108,88.09,-56.8237,9E+09,9E+09,9E+09]], v200, z50, tPKI500\WObj:=w7000714;
MoveJ [[725.96,833.32,299.94],[0.949488,0.0555833,-0.136527,0.277028],[0,-1,0,0],[413.553,106.616,-53.5223,9E+09,9E+09,9E+09]], v200, z50, tPKI500\WObj:=w7000714;
ArcLStart [[807.48,733.81,271.76],[0.939491,0.307711,-0.0100868,0.150235],[0,-1,0,0],[413.565,106.616,-53.5265,9E+09,9E+09,9E+09]], v200, seam1, m178job76, fine, tPKI500\WObj:=w7000714;
ArcL [[760.43,775.23,297.72],[0.926981,0.356956,0.0319106,0.110776],[0,0,0,0],[413.548,106.616,-53.5247,9E+09,9E+09,9E+09]], v200, seam1, m178job76, z50, tPKI500\WObj:=w7000714;
ArcL [[760.07,777.51,303.26],[0.698169,0.649358,0.242999,-0.17846],[0,0,-1,0],[413.543,106.616,-53.5239,9E+09,9E+09,9E+09]], v200, seam1, m178job76, z50, tPKI500\WObj:=w7000714;
ArcL [[871.56,777.98,519.92],[0.57154,0.700451,0.323416,-0.279487],[1,0,-1,0],[413.551,106.616,-53.5251,9E+09,9E+09,9E+09]], v200, seam1, m178job76, z50, tPKI500\WObj:=w7000714;
ArcL [[877.73,774.28,523.84],[0.040511,0.71107,0.485785,-0.506707],[1,0,-2,0],[413.551,106.616,-53.5247,9E+09,9E+09,9E+09]], v200, seam1, m178job76, z10, tPKI500\WObj:=w7000714;
ArcL [[923.64,733.95,501.06],[0.0676337,-0.67985,-0.496463,0.535496],[1,0,-2,0],[413.546,106.616,-53.5247,9E+09,9E+09,9E+09]], v200, seam1, m178job76, z10, tPKI500\WObj:=w7000714;
ArcL [[925.38,729.96,494.21],[0.618752,-0.34959,-0.431571,0.55559],[1,-1,-3,0],[413.551,106.616,-53.5239,9E+09,9E+09,9E+09]], v200, seam1, m178job76, z50, tPKI500\WObj:=w7000714;
ArcLEnd [[813.74,731.41,274.30],[0.705757,-0.211786,-0.442513,0.511114],[1,-1,-3,0],[413.551,106.616,-53.5247,9E+09,9E+09,9E+09]], v200, seam1, m178job76, fine, tPKI500\WObj:=w7000714;
MoveJ [[908.61,863.35,230.68],[0.813108,-0.10966,-0.322805,0.471835],[1,-1,-3,0],[413.552,106.616,-53.524,9E+09,9E+09,9E+09]], v600, z50, tPKI500\WObj:=w7000714;


MoveJ mooduli_vahetus, v200, z50, tPKI500\WObj:=w7000714;

ENDPROC


  PROC PuhdistRutWeld()
   MoveJ pHomeS2, v500, fine, tPKI500;
   DeactUnit STN2;
   %"puhdistaa"%;
   ActUnit STN2;
   MoveJ pHomeS2, v500, fine, tPKI500;
  ENDPROC


ENDMODULE
